(* CoDeSys 2.3.9.25 project: Michal.pro *)
(* Libraries: Standard.lib 22.11.04 11:21:12, SYSLIBCALLBACK.LIB 20.4.05 11:04:48 *)

(* PLC configuration (modules and I/O channels)
out1 AT %QX4.0 [BOOLOnX_Q] Ch_1 Digital output
out2 AT %QX4.1 [BOOLOnX_Q] Ch_2 Digital output
out3 AT %QX4.2 [BOOLOnX_Q] Ch_1 Digital output
out4 AT %QX4.3 [BOOLOnX_Q] Ch_2 Digital output
out5 AT %QX4.4 [BOOLOnX_Q] Ch_3 Digital output
out6 AT %QX4.5 [BOOLOnX_Q] Ch_4 Digital output
out7 AT %QX4.6 [BOOLOnX_Q] Ch_5 Digital output
out8 AT %QX4.7 [BOOLOnX_Q] Ch_6 Digital output
out9 AT %QX4.8 [BOOLOnX_Q] Ch_7 Digital output
out10 AT %QX4.9 [BOOLOnX_Q] Ch_8 Digital output
in1 AT %IX8.0 [BOOLOnX_I] Ch_1 Digital input
in2 AT %IX8.1 [BOOLOnX_I] Ch_2 Digital input
in3 AT %IX8.2 [BOOLOnX_I] Ch_3 Digital input
in4 AT %IX8.3 [BOOLOnX_I] Ch_4 Digital input
in5 AT %IX8.4 [BOOLOnX_I] Ch_5 Digital input
in6 AT %IX8.5 [BOOLOnX_I] Ch_6 Digital input
in7 AT %IX8.6 [BOOLOnX_I] Ch_7 Digital input
in8 AT %IX8.7 [BOOLOnX_I] Ch_8 Digital input
0750-0430 8 DI 24 V DC 3.0ms [Type_1_8_Channels] node 0, in %IB0 out %QB0 {INTTypePAAssignment = PLC; INTTypeModule = plugged}
  AT %IX8.8 [BOOLOnX_I] Ch_1 Digital input
  AT %IX8.9 [BOOLOnX_I] Ch_2 Digital input
  AT %IX8.10 [BOOLOnX_I] Ch_3 Digital input
  AT %IX8.11 [BOOLOnX_I] Ch_4 Digital input
  AT %IX8.12 [BOOLOnX_I] Ch_5 Digital input
  AT %IX8.13 [BOOLOnX_I] Ch_6 Digital input
  AT %IX8.14 [BOOLOnX_I] Ch_7 Digital input
  AT %IX8.15 [BOOLOnX_I] Ch_8 Digital input
teplota1 AT %IW0 [INTOnW_I] Ch_1 signed Input value
teplota2 AT %IW1 [INTOnW_I] Ch_2 signed Input value
teplota3 AT %IW2 [INTOnW_I] Ch_3 signed Input value
teplota4 AT %IW3 [INTOnW_I] Ch_4 signed Input value
0750-0559 4 AO 0-10V DC [Type_14_4_Channels] node 0, in %IB0 out %QB0 {INTTypePAAssignment = PLC; INTTypeModule = plugged}
  AT %QW0 [WORDOnW_Q] Ch_1 Analog output
  AT %QW1 [WORDOnW_Q] Ch_2 Analog output
  AT %QW2 [WORDOnW_Q] Ch_3 Analog output
  AT %QW3 [WORDOnW_Q] Ch_4 Analog output
0750-0455 4 AI 4-20mA s.e. [Type_8_4_Channels] node 0, in %IB0 out %QB0 {INTTypePAAssignment = PLC; INTTypeModule = plugged}
  AT %IW4 [WORDOnW_I] Ch_1 Input word
  AT %IW5 [WORDOnW_I] Ch_2 Input word
  AT %IW6 [WORDOnW_I] Ch_3 Input word
  AT %IW7 [WORDOnW_I] Ch_4 Input word
Fieldbus variables [FB_VARS] node 1, in %IB0 out %QB0
*)

(* POU PLC_PRG, LD *)
PROGRAM PLC_PRG
VAR
END_VAR
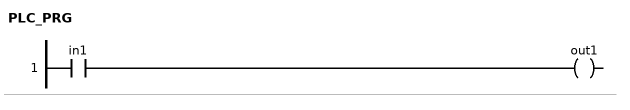
_LD_ (* Ladder Diagram *)
NETWORK 1
	[in1] --- (out1)
_END_LD_
(* the same logic as Structured Text *)
(* Network 1 *)
out1 := in1;
END_PROGRAM
